{attribute 'qualified_only'}
{attribute 'strict'}
TYPE eSupportedHeatpumps :
(
	TranePicco := 0,
	LgThermaV	:= 1
);
END_TYPE

(* stored: Version 1.1.0.1, ProductVersion 3.1.4026.18
   DUT eSupportedHeatpumps: Id {435fcd2f-8102-4844-91c6-846f2f9ea814} *)
